(* Logix 5000 project; controller cal1615 1756-L62 rev 20.19; software revision 20.05; part 15 of 81 *)
(* tags used below, declared in another part *)
   FAULT : BOOL;   // Fault AFI
   p01_r15_footage_ft : REAL;   // System Customer Footage Counter
   p01_real_to_hmi : REAL[112];   // System Real to HMI
   p01r09_pb_global_reset : BOOL;   // System Modes PB: Global Fault Reset
   p02_real_to_hmi : hmi_real;   // MOP HMI Iface Real to HMI
   p02r01 : routine;   // MOP HMI Iface Main
   p02r06 : routine;   // MOP HMI Iface Real to HMI
   p02r06_timer_fault : TIMER[4];   // MOP HMI Iface Real to HMI Fault Delay
   p02r06_timer_warning : TIMER[4];   // MOP HMI Iface Real to HMI Warning Delay
   p02r07 : routine;   // MOP HMI Iface Alarms
   p02r07_timer_fault : TIMER[4];   // MOP HMI Iface Alarms Fault Delay
   p02r07_timer_warning : TIMER[4];   // MOP HMI Iface Alarms Warning Delay
   p02r08 : routine;   // MOP HMI Iface Warnings
   p02r08_timer_fault : TIMER[4];   // MOP HMI Iface Warnings Fault Delay
   p02r08_timer_warning : TIMER[4];   // MOP HMI Iface Warnings Warning Delay
   p02r09 : routine;   // MOP HMI Iface Maintenance
   p02r09_timer_fault : TIMER[4];   // MOP HMI Iface Maintenance Fault Delay
   p02r09_timer_warning : TIMER[4];   // MOP HMI Iface Maintenance Warning Delay
   p02r10 : routine;   // MOP HMI Iface
   p02r10_timer_fault : TIMER[4];   // MOP HMI Iface Fault Delay
   p02r10_timer_warning : TIMER[4];   // MOP HMI Iface Warning Delay
   p11_real_to_hmi : REAL[112];   // Zone 1 Real to HMI
   p12_real_to_hmi : REAL[112];   // Zone 2 Real to HMI
   p13_real_to_hmi : REAL[112];   // Zone 3 Real to HMI
   p19_real_to_hmi : REAL[80];   // Advanced Cooling Real to HMI
   p20_real_to_hmi : REAL[112];   // Letoff Real to HMI
   p21_real_to_hmi : REAL[112];   // Splice Press Real to HMI
   p22_real_to_hmi : REAL[112];   // Tension Stand 1 Real to HMI
   p23_real_to_hmi : REAL[112];   // Impreg Real to HMI
   p24_real_to_hmi : REAL[112];   // Tension Stand 2 Real to HMI
   p25_real_to_hmi : REAL[112];   // Tension Stand 2 Real to HMI
   p26_real_to_hmi : REAL[112];   // Lower Poly Letoff Real to HMI
   p27_real_to_hmi : REAL[112];   // Winder Real to HMI
   p28_real_to_hmi : REAL[112];
   p29_real_to_hmi : REAL[112];   // Laminator Real to HMI
(* P02_MOP_HMI_Iface, continued *)

ROUTINE R06_Real_to_HMI   (* ladder *)
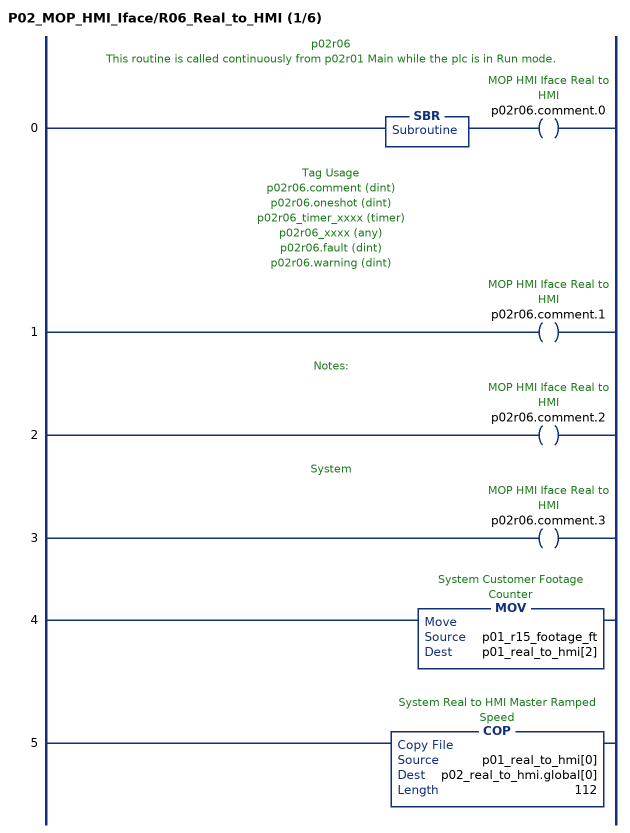
   // p02r06
   // This routine is called continuously from p02r01 Main while the plc is in Run mode.
   0: SBR()OTE(p02r06.comment.0);
   // Tag Usage
   // p02r06.comment (dint)
   // p02r06.oneshot (dint)
   // p02r06_timer_xxxx (timer)
   // p02r06_xxxx (any)
   // p02r06.fault (dint)
   // p02r06.warning (dint)
   1: OTE(p02r06.comment.1);
   // Notes:
   2: OTE(p02r06.comment.2);
   // System
   3: OTE(p02r06.comment.3);
   4: MOV(p01_r15_footage_ft,p01_real_to_hmi[2]);
   5: COP(p01_real_to_hmi[0],p02_real_to_hmi.global[0],112);
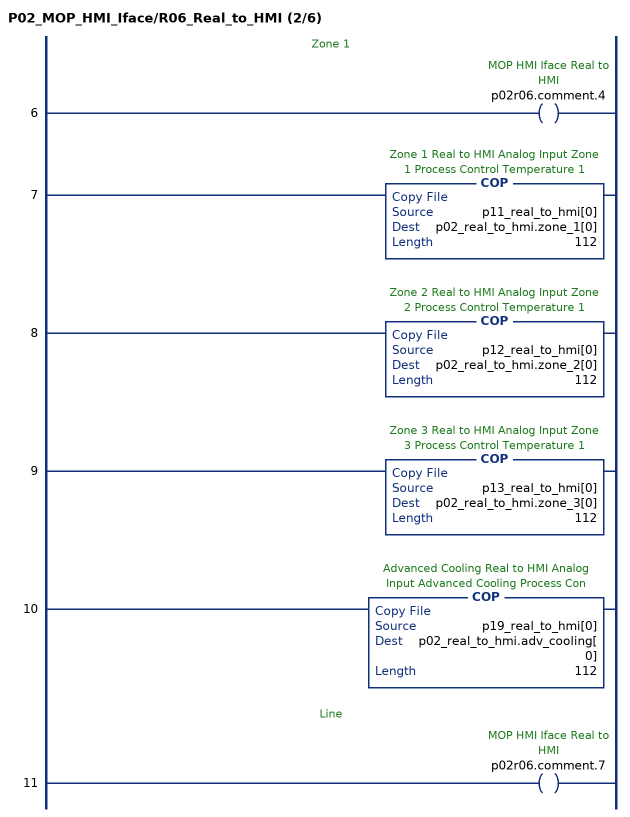
   // Zone 1
   6: OTE(p02r06.comment.4);
   7: COP(p11_real_to_hmi[0],p02_real_to_hmi.zone_1[0],112);
   8: COP(p12_real_to_hmi[0],p02_real_to_hmi.zone_2[0],112);
   9: COP(p13_real_to_hmi[0],p02_real_to_hmi.zone_3[0],112);
   10: COP(p19_real_to_hmi[0],p02_real_to_hmi.adv_cooling[0],112);
   // Line
   11: OTE(p02r06.comment.7);
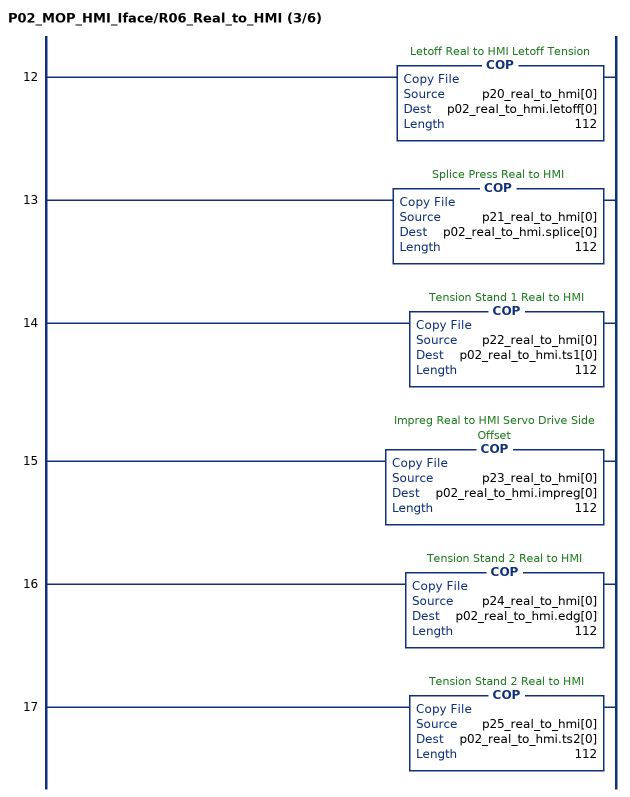
   12: COP(p20_real_to_hmi[0],p02_real_to_hmi.letoff[0],112);
   13: COP(p21_real_to_hmi[0],p02_real_to_hmi.splice[0],112);
   14: COP(p22_real_to_hmi[0],p02_real_to_hmi.ts1[0],112);
   15: COP(p23_real_to_hmi[0],p02_real_to_hmi.impreg[0],112);
   16: COP(p24_real_to_hmi[0],p02_real_to_hmi.edg[0],112);
   17: COP(p25_real_to_hmi[0],p02_real_to_hmi.ts2[0],112);
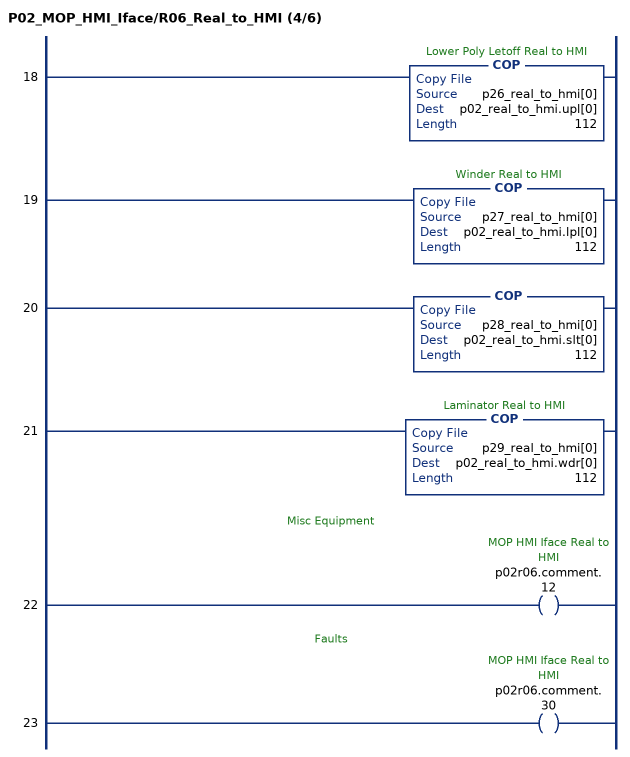
   18: COP(p26_real_to_hmi[0],p02_real_to_hmi.upl[0],112);
   19: COP(p27_real_to_hmi[0],p02_real_to_hmi.lpl[0],112);
   20: COP(p28_real_to_hmi[0],p02_real_to_hmi.slt[0],112);
   21: COP(p29_real_to_hmi[0],p02_real_to_hmi.wdr[0],112);
   // Misc Equipment
   22: OTE(p02r06.comment.12);
   // Faults
   23: OTE(p02r06.comment.30);
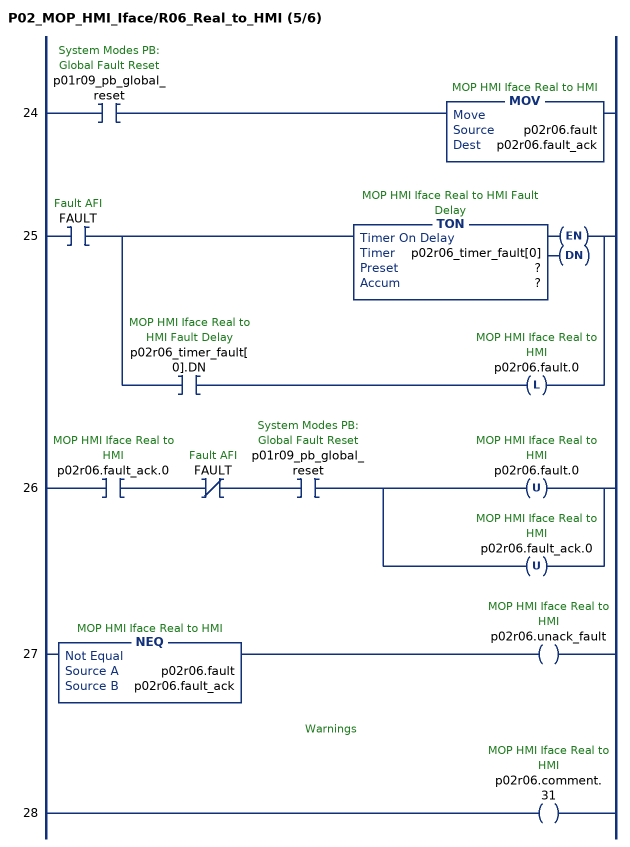
   24: XIC(p01r09_pb_global_reset)MOV(p02r06.fault,p02r06.fault_ack);
   25: XIC(FAULT)[TON(p02r06_timer_fault[0],?,?) ,XIC(p02r06_timer_fault[0].DN) OTL(p02r06.fault.0) ];
   26: XIC(p02r06.fault_ack.0)XIO(FAULT)XIC(p01r09_pb_global_reset)[OTU(p02r06.fault.0) ,OTU(p02r06.fault_ack.0) ];
   27: NEQ(p02r06.fault,p02r06.fault_ack)OTE(p02r06.unack_fault);
   // Warnings
   28: OTE(p02r06.comment.31);
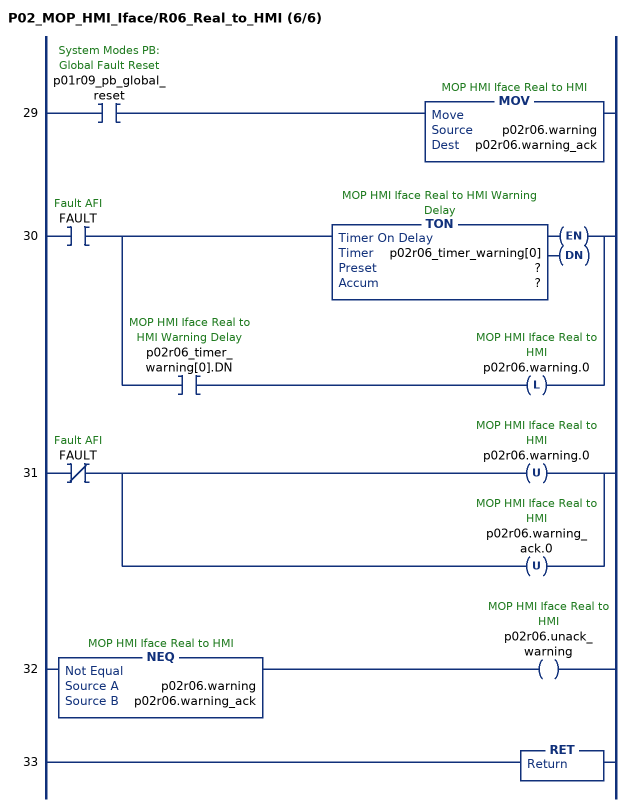
   29: XIC(p01r09_pb_global_reset)MOV(p02r06.warning,p02r06.warning_ack);
   30: XIC(FAULT)[TON(p02r06_timer_warning[0],?,?) ,XIC(p02r06_timer_warning[0].DN) OTL(p02r06.warning.0) ];
   31: XIO(FAULT)[OTU(p02r06.warning.0) ,OTU(p02r06.warning_ack.0) ];
   32: NEQ(p02r06.warning,p02r06.warning_ack)OTE(p02r06.unack_warning);
   33: RET();
END_ROUTINE

ROUTINE R07_Alarms   (* ladder *)
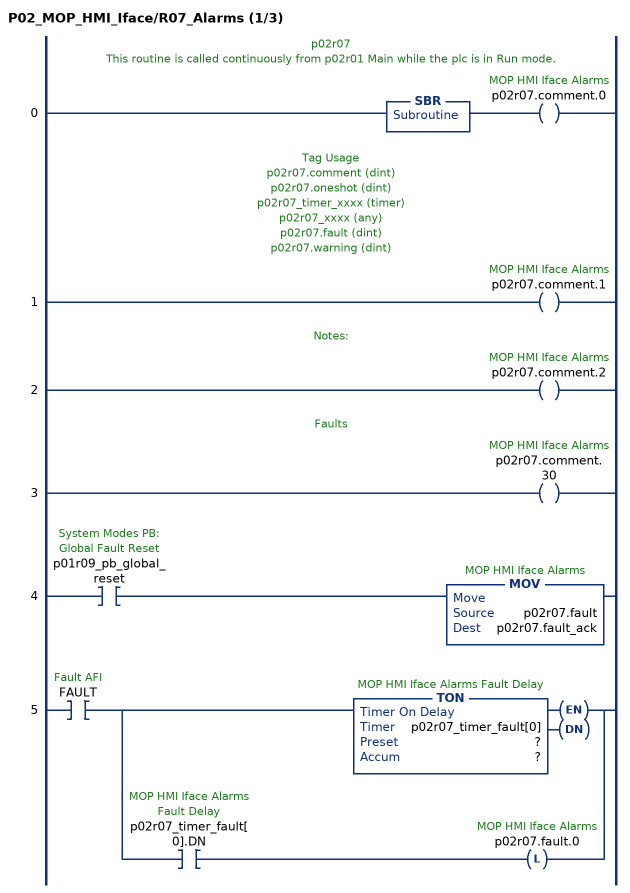
   // p02r07
   // This routine is called continuously from p02r01 Main while the plc is in Run mode.
   0: SBR()OTE(p02r07.comment.0);
   // Tag Usage
   // p02r07.comment (dint)
   // p02r07.oneshot (dint)
   // p02r07_timer_xxxx (timer)
   // p02r07_xxxx (any)
   // p02r07.fault (dint)
   // p02r07.warning (dint)
   1: OTE(p02r07.comment.1);
   // Notes:
   2: OTE(p02r07.comment.2);
   // Faults
   3: OTE(p02r07.comment.30);
   4: XIC(p01r09_pb_global_reset)MOV(p02r07.fault,p02r07.fault_ack);
   5: XIC(FAULT)[TON(p02r07_timer_fault[0],?,?) ,XIC(p02r07_timer_fault[0].DN) OTL(p02r07.fault.0) ];
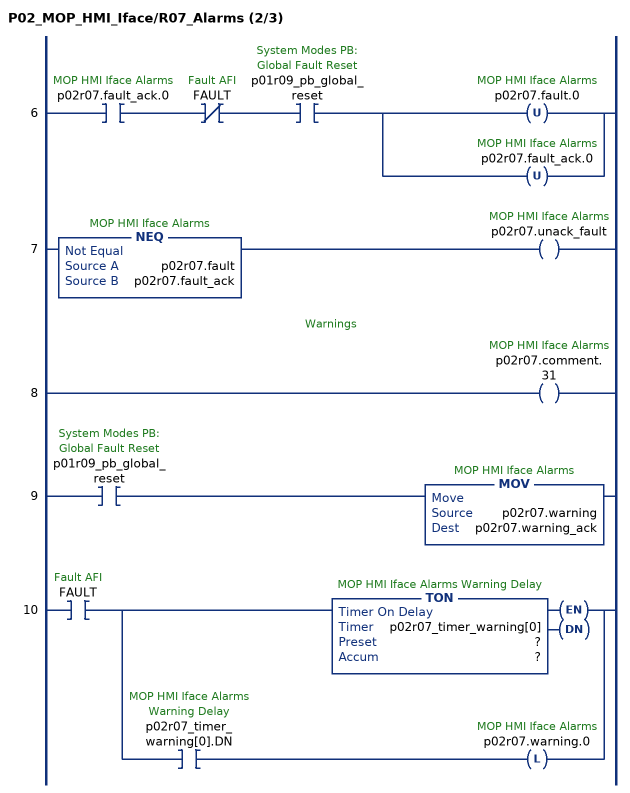
   6: XIC(p02r07.fault_ack.0)XIO(FAULT)XIC(p01r09_pb_global_reset)[OTU(p02r07.fault.0) ,OTU(p02r07.fault_ack.0) ];
   7: NEQ(p02r07.fault,p02r07.fault_ack)OTE(p02r07.unack_fault);
   // Warnings
   8: OTE(p02r07.comment.31);
   9: XIC(p01r09_pb_global_reset)MOV(p02r07.warning,p02r07.warning_ack);
   10: XIC(FAULT)[TON(p02r07_timer_warning[0],?,?) ,XIC(p02r07_timer_warning[0].DN) OTL(p02r07.warning.0) ];
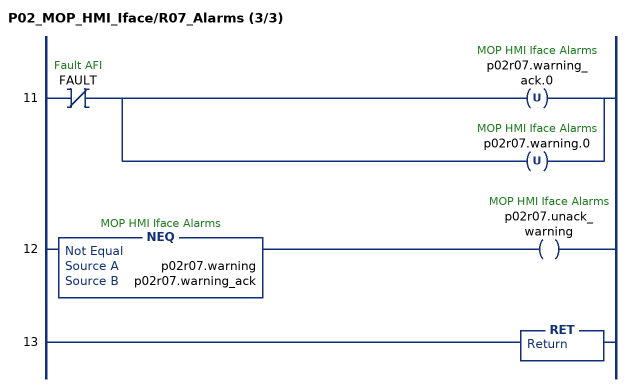
   11: XIO(FAULT)[OTU(p02r07.warning_ack.0) ,OTU(p02r07.warning.0) ];
   12: NEQ(p02r07.warning,p02r07.warning_ack)OTE(p02r07.unack_warning);
   13: RET();
END_ROUTINE

ROUTINE R08_Warnings   (* ladder *)
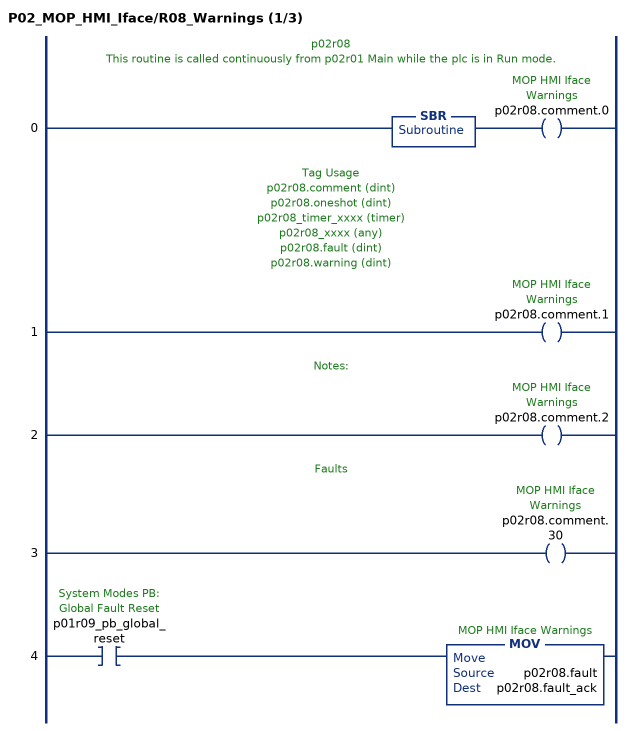
   // p02r08
   // This routine is called continuously from p02r01 Main while the plc is in Run mode.
   0: SBR()OTE(p02r08.comment.0);
   // Tag Usage
   // p02r08.comment (dint)
   // p02r08.oneshot (dint)
   // p02r08_timer_xxxx (timer)
   // p02r08_xxxx (any)
   // p02r08.fault (dint)
   // p02r08.warning (dint)
   1: OTE(p02r08.comment.1);
   // Notes:
   2: OTE(p02r08.comment.2);
   // Faults
   3: OTE(p02r08.comment.30);
   4: XIC(p01r09_pb_global_reset)MOV(p02r08.fault,p02r08.fault_ack);
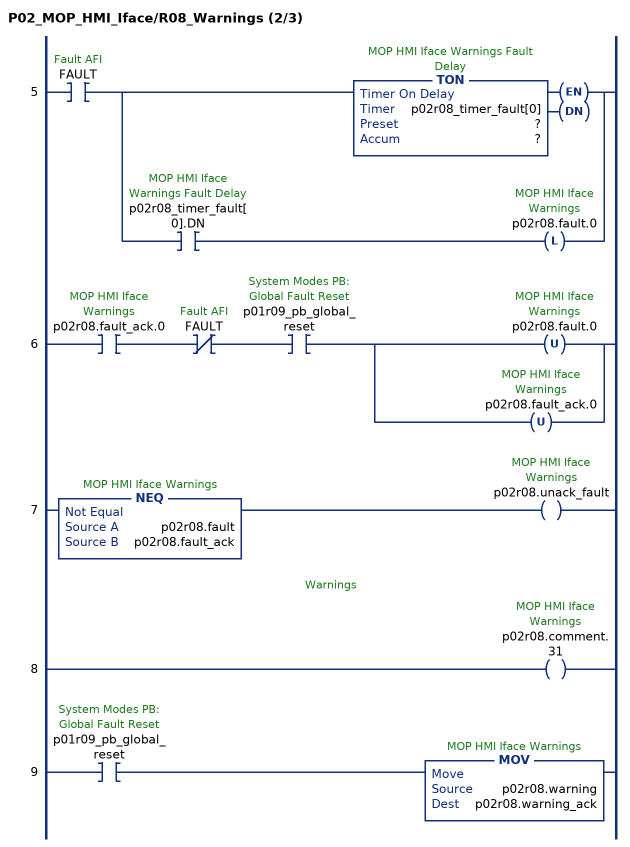
   5: XIC(FAULT)[TON(p02r08_timer_fault[0],?,?) ,XIC(p02r08_timer_fault[0].DN) OTL(p02r08.fault.0) ];
   6: XIC(p02r08.fault_ack.0)XIO(FAULT)XIC(p01r09_pb_global_reset)[OTU(p02r08.fault.0) ,OTU(p02r08.fault_ack.0) ];
   7: NEQ(p02r08.fault,p02r08.fault_ack)OTE(p02r08.unack_fault);
   // Warnings
   8: OTE(p02r08.comment.31);
   9: XIC(p01r09_pb_global_reset)MOV(p02r08.warning,p02r08.warning_ack);
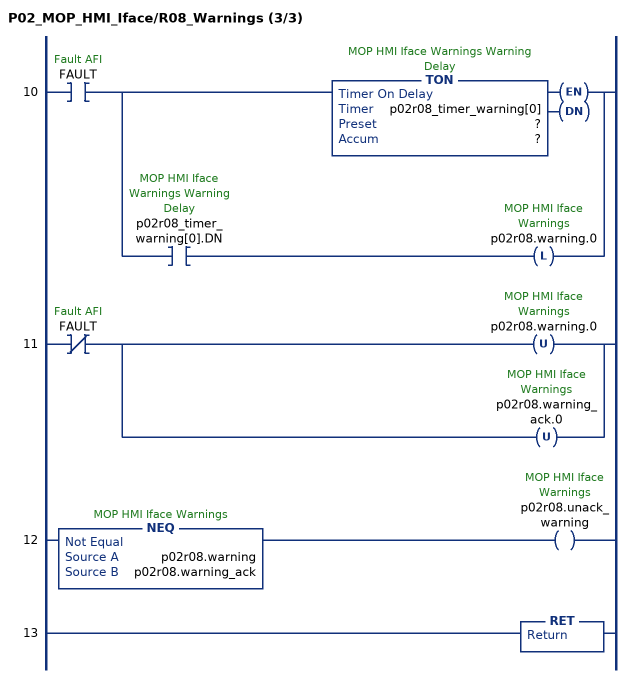
   10: XIC(FAULT)[TON(p02r08_timer_warning[0],?,?) ,XIC(p02r08_timer_warning[0].DN) OTL(p02r08.warning.0) ];
   11: XIO(FAULT)[OTU(p02r08.warning.0) ,OTU(p02r08.warning_ack.0) ];
   12: NEQ(p02r08.warning,p02r08.warning_ack)OTE(p02r08.unack_warning);
   13: RET();
END_ROUTINE

ROUTINE R09_Maintenance   (* ladder *)
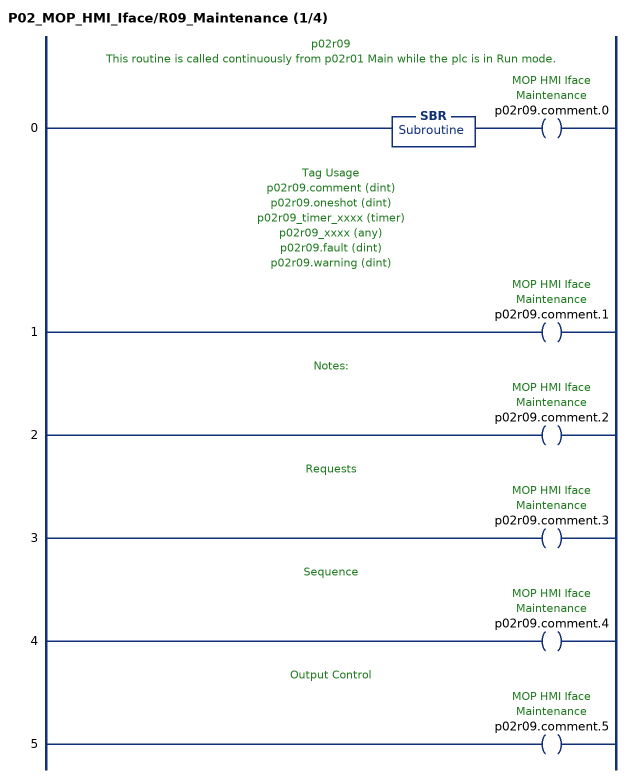
   // p02r09
   // This routine is called continuously from p02r01 Main while the plc is in Run mode.
   0: SBR()OTE(p02r09.comment.0);
   // Tag Usage
   // p02r09.comment (dint)
   // p02r09.oneshot (dint)
   // p02r09_timer_xxxx (timer)
   // p02r09_xxxx (any)
   // p02r09.fault (dint)
   // p02r09.warning (dint)
   1: OTE(p02r09.comment.1);
   // Notes:
   2: OTE(p02r09.comment.2);
   // Requests
   3: OTE(p02r09.comment.3);
   // Sequence
   4: OTE(p02r09.comment.4);
   // Output Control
   5: OTE(p02r09.comment.5);
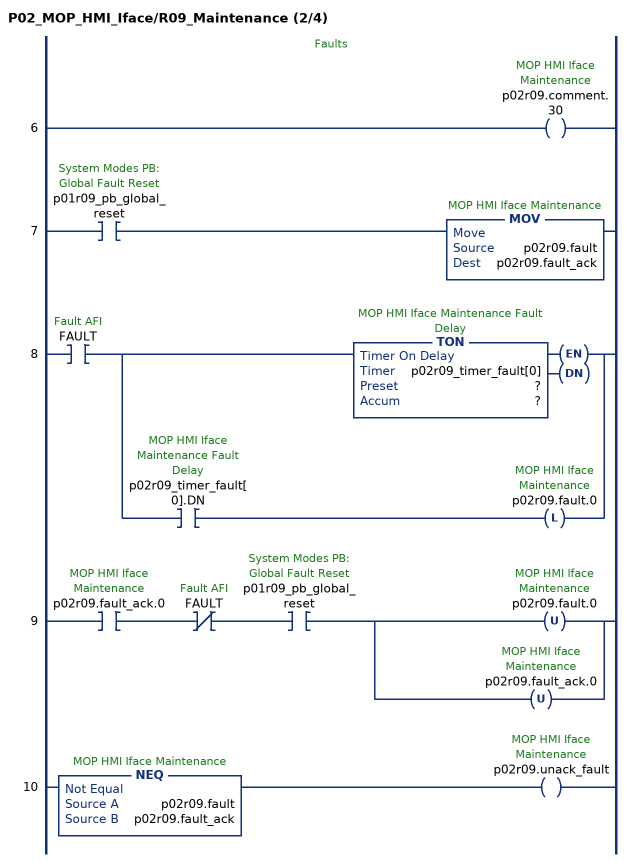
   // Faults
   6: OTE(p02r09.comment.30);
   7: XIC(p01r09_pb_global_reset)MOV(p02r09.fault,p02r09.fault_ack);
   8: XIC(FAULT)[TON(p02r09_timer_fault[0],?,?) ,XIC(p02r09_timer_fault[0].DN) OTL(p02r09.fault.0) ];
   9: XIC(p02r09.fault_ack.0)XIO(FAULT)XIC(p01r09_pb_global_reset)[OTU(p02r09.fault.0) ,OTU(p02r09.fault_ack.0) ];
   10: NEQ(p02r09.fault,p02r09.fault_ack)OTE(p02r09.unack_fault);
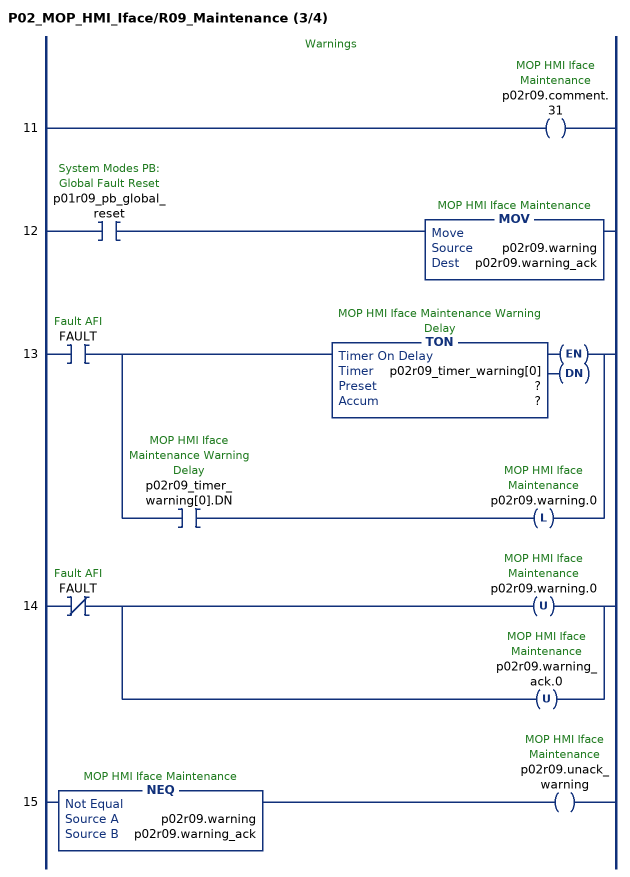
   // Warnings
   11: OTE(p02r09.comment.31);
   12: XIC(p01r09_pb_global_reset)MOV(p02r09.warning,p02r09.warning_ack);
   13: XIC(FAULT)[TON(p02r09_timer_warning[0],?,?) ,XIC(p02r09_timer_warning[0].DN) OTL(p02r09.warning.0) ];
   14: XIO(FAULT)[OTU(p02r09.warning.0) ,OTU(p02r09.warning_ack.0) ];
   15: NEQ(p02r09.warning,p02r09.warning_ack)OTE(p02r09.unack_warning);
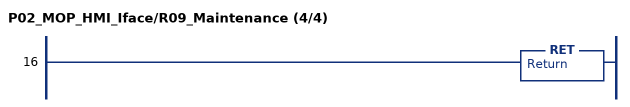
   16: RET();
END_ROUTINE

ROUTINE R10   (* ladder *)
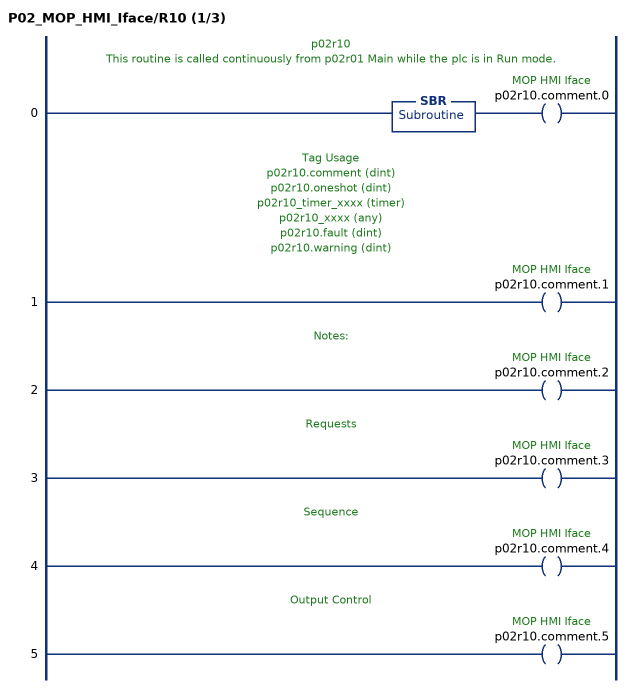
   // p02r10
   // This routine is called continuously from p02r01 Main while the plc is in Run mode.
   0: SBR()OTE(p02r10.comment.0);
   // Tag Usage
   // p02r10.comment (dint)
   // p02r10.oneshot (dint)
   // p02r10_timer_xxxx (timer)
   // p02r10_xxxx (any)
   // p02r10.fault (dint)
   // p02r10.warning (dint)
   1: OTE(p02r10.comment.1);
   // Notes:
   2: OTE(p02r10.comment.2);
   // Requests
   3: OTE(p02r10.comment.3);
   // Sequence
   4: OTE(p02r10.comment.4);
   // Output Control
   5: OTE(p02r10.comment.5);
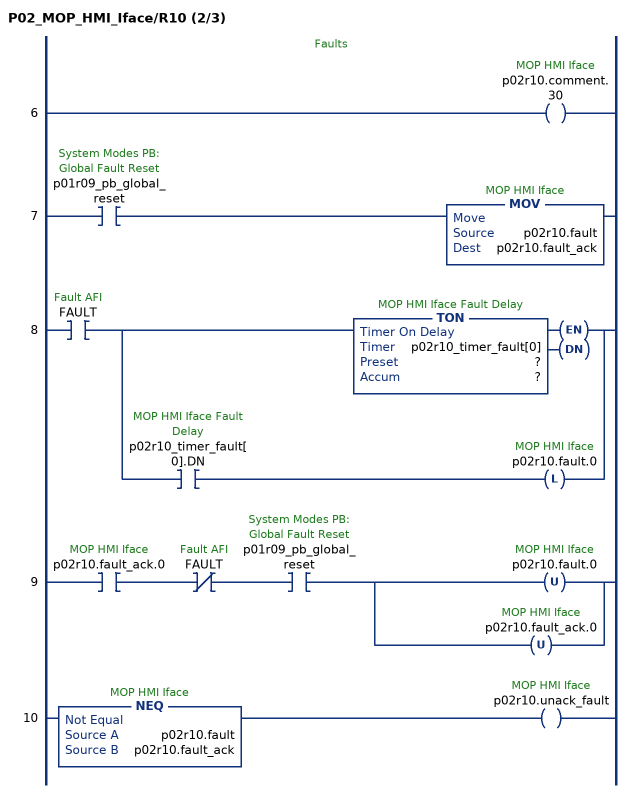
   // Faults
   6: OTE(p02r10.comment.30);
   7: XIC(p01r09_pb_global_reset)MOV(p02r10.fault,p02r10.fault_ack);
   8: XIC(FAULT)[TON(p02r10_timer_fault[0],?,?) ,XIC(p02r10_timer_fault[0].DN) OTL(p02r10.fault.0) ];
   9: XIC(p02r10.fault_ack.0)XIO(FAULT)XIC(p01r09_pb_global_reset)[OTU(p02r10.fault.0) ,OTU(p02r10.fault_ack.0) ];
   10: NEQ(p02r10.fault,p02r10.fault_ack)OTE(p02r10.unack_fault);
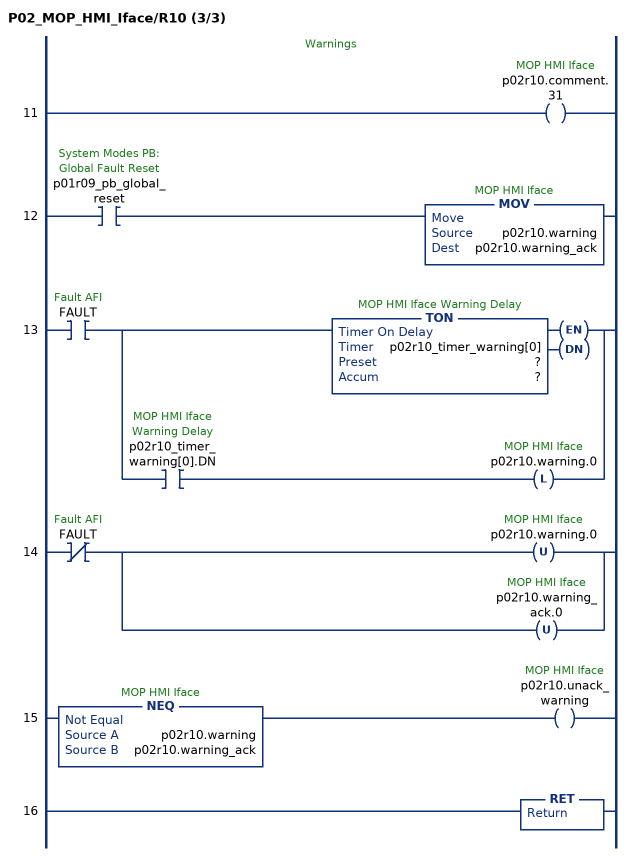
   // Warnings
   11: OTE(p02r10.comment.31);
   12: XIC(p01r09_pb_global_reset)MOV(p02r10.warning,p02r10.warning_ack);
   13: XIC(FAULT)[TON(p02r10_timer_warning[0],?,?) ,XIC(p02r10_timer_warning[0].DN) OTL(p02r10.warning.0) ];
   14: XIO(FAULT)[OTU(p02r10.warning.0) ,OTU(p02r10.warning_ack.0) ];
   15: NEQ(p02r10.warning,p02r10.warning_ack)OTE(p02r10.unack_warning);
   16: RET();
END_ROUTINE
